(* IEC 61131-3 sources: AXOpen/src/integrations/app/src/Examples/AXOpen.AxoData, 8 files *)

(* ---- AxoDataDocuExample.st ---- *)
USING AXOpen.Core;
using AXOpen.Data;

NAMESPACE AxoDataExamplesDocu

    //<ProcessDataMangerDeclaration>
    {S7.extern=ReadWrite}
    CLASS AxoProcessDataManager EXTENDS AXOpen.Data.AxoDataExchange
        VAR PUBLIC
            {#ix-generic:TOnline}
            {#ix-generic:TPlain as POCO}
            {#ix-attr:[AxoDataEntityAttribute]}
            Data       : AxoProductionData;    // <-  Manager will operate on this member.
        END_VAR
    END_CLASS
    //</ProcessDataMangerDeclaration>

    //<ProcessDataDeclaration>
    {S7.extern=ReadWrite}
    CLASS AxoProductionData EXTENDS AXOpen.Data.AxoDataEntity
        VAR PUBLIC
            {#ix-set:AttributeName = "Some string data"}
            SomeData : STRING;
            {#ix-set:AttributeName = "Some number"}
            SomeNumber : INT;
            {#ix-set:AttributeName = "Some boolean"}
            SomeBool : BOOL;
        END_VAR
    END_CLASS
    //</ProcessDataDeclaration>

    //<ContextDeclaration>
    {S7.extern=ReadWrite}
    CLASS PUBLIC Context EXTENDS AXOpen.Core.AxoContext
        VAR PUBLIC
            DataManager : AxoProcessDataManager;
            _rootObject :   AxoObject;
        END_VAR

        METHOD OVERRIDE Main
            THIS.InitializeRootObject(_rootObject);
            DataManager.Run(_rootObject);
        END_METHOD
    END_CLASS
    //</ContextDeclaration>

    //<UseManager>
    {S7.extern=ReadWrite}
    CLASS UseManager
        VAR
            _create : BOOL;
            _read : BOOL;
            _update : BOOL;
            _delete : BOOL;
            _id : STRING;
        END_VAR

        METHOD Use
            VAR_IN_OUT
                DataManager : AxoProcessDataManager;
            END_VAR
            IF(_create) THEN
                IF(DataManager.Create(_id).IsDone()) THEN
                    _create := FALSE;
                END_IF;
            END_IF;

            IF(_read) THEN
                IF(DataManager.Read(_id).IsDone()) THEN
                    _read := FALSE;
                END_IF;
            END_IF;

            IF(_update) THEN
                IF(DataManager.Update(_id).IsDone()) THEN
                    _update := FALSE;
                END_IF;
            END_IF;

            IF(_delete) THEN
                IF(DataManager.Delete(_id).IsDone()) THEN
                    _delete := FALSE;
                END_IF;
            END_IF;
        END_METHOD
    END_CLASS
    //</UseManager>

END_NAMESPACE

(* ---- AxoDataFragmentExchangeDocu.st ---- *)
USING AXOpen.Core;
USING AXOpen.Data;
USING AXOpen.Probers;

NAMESPACE AxoDataFramentsExchangeDocuExample

    //<ContextDeclaration>
    {S7.extern=ReadWrite}
    CLASS AxoDataFragmentExchangeContext EXTENDS AXOpen.Core.AxoContext
        VAR PUBLIC
            ProcessData : ProcessDataManager;
            _rootObject :   AxoObject;
        END_VAR

        METHOD PROTECTED OVERRIDE Main
            _rootObject.InitializeWithContext(THIS);
            // This is required to run cyclically. Method provides handling of data exchange tasks.
            ProcessData.Run(_rootObject);
        END_METHOD
    END_CLASS
    //</ContextDeclaration>

    //<ProcessDataMangerDeclaration>
    {S7.extern=ReadWrite}
    CLASS ProcessDataManager EXTENDS AXOpen.Data.AxoDataFragmentExchange
        VAR PUBLIC
            {#ix-attr:[AXOpen.Data.AxoDataFragmentAttribute]}
            SharedHeader : SharedDataHeaderManger;
            {#ix-attr:[AXOpen.Data.AxoDataFragmentAttribute]}
            Station_1 : Station_1_ProcessDataManger;
        END_VAR
    END_CLASS
    //</ProcessDataMangerDeclaration>

     //<UseManager>
     {S7.extern=ReadWrite}
     CLASS UseManager
        VAR
            _create : BOOL;
            _read : BOOL;
            _update : BOOL;
            _delete : BOOL;
            _id : STRING;
        END_VAR

        METHOD Use
            VAR_IN_OUT
                DataFragmentManager : ProcessDataManager;
            END_VAR
            IF(_create) THEN
                IF(DataFragmentManager.Create(_id).IsDone()) THEN
                    _create := FALSE;
                END_IF;
            END_IF;

            IF(_read) THEN
                IF(DataFragmentManager.Read(_id).IsDone()) THEN
                    _read := FALSE;
                END_IF;
            END_IF;

            IF(_update) THEN
                IF(DataFragmentManager.Update(_id).IsDone()) THEN
                    _update := FALSE;
                END_IF;
            END_IF;

            IF(_delete) THEN
                IF(DataFragmentManager.Delete(_id).IsDone()) THEN
                    _delete := FALSE;
                END_IF;
            END_IF;
        END_METHOD
    END_CLASS
    //</UseManager>

    {S7.extern=ReadWrite}
    CLASS SharedDataHeaderData EXTENDS AXOpen.Data.AxoDataEntity
        VAR PUBLIC
            {#ix-set:AttributeName = "Some string data"}
            SomeData : STRING;
            {#ix-set:AttributeName = "Some number"}
            SomeNumber : INT;
            {#ix-set:AttributeName = "Some boolean"}
            SomeBool : BOOL;
        END_VAR
    END_CLASS

    {S7.extern=ReadWrite}
    CLASS SharedDataHeaderManger EXTENDS AXOpen.Data.AxoDataExchange
        VAR PUBLIC
            {#ix-generic:TOnline}
            {#ix-generic:TPlain as POCO}
            {#ix-attr:[AXOpen.Data.AxoDataEntityAttribute]}
            {#ix-attr:[Container(Layout.Stack)]}
            {#ix-set:AttributeName = "Shared Header"}
            Set : SharedDataHeaderData;
        END_VAR
    END_CLASS

    {S7.extern=ReadWrite}
    CLASS Station_1_ProcessDataManger
        EXTENDS AXOpen.Data.AxoDataExchange
        VAR PUBLIC
            {#ix-generic:TOnline}
            {#ix-generic:TPlain as POCO}
            {#ix-attr:[AXOpen.Data.AxoDataEntityAttribute]}
            {#ix-attr:[Container(Layout.Stack)]}
            {#ix-set:AttributeName = "Station 1"}
            Set : Station_1_Data;
        END_VAR
    END_CLASS

    {S7.extern=ReadWrite}
    CLASS Station_1_Data
        EXTENDS AXOpen.Data.AxoDataEntity
        VAR PUBLIC
            {#ix-set:AttributeName = "Some string data"}
            SomeData : STRING;
            {#ix-set:AttributeName = "Some number"}
            SomeNumber : INT;
            {#ix-set:AttributeName = "Some boolean"}
            SomeBool : BOOL;
        END_VAR
    END_CLASS
END_NAMESPACE

(* ---- AxoProcessDataManager.st ---- *)
using AXOpen.Data;

NAMESPACE AxoDataExamples

    CLASS AxoProcessDataManager EXTENDS AXOpen.Data.AxoDataExchange
        VAR PUBLIC
            _identifier : STRING;
            _create     : BOOL;
            _read       : BOOL;
            _update     : BOOL;
            _delete     : BOOL;
            {#ix-generic:TOnline}
            {#ix-generic:TPlain as POCO}
            {#ix-attr:[AxoDataEntityAttribute]}
            _data       : AxoProductionData;
            // _data       : AxoProductionDataInherited;
        END_VAR
    END_CLASS
END_NAMESPACE

(* ---- AxoProductionData.st ---- *)
using AXOpen.Data;

NAMESPACE AxoDataExamples

    CLASS AxoProductionData EXTENDS AXOpen.Data.AxoDataEntity
        VAR PUBLIC
            RecipeName : STRING;
        END_VAR
    END_CLASS

END_NAMESPACE

(* ---- AxoProductionDataInherited.st ---- *)
using AXOpen.Data;

NAMESPACE AxoDataExamples

    {S7.extern=ReadWrite}
    CLASS AxoProductionDataInherited EXTENDS AxoProductionData
        VAR PUBLIC
            RecipeName2 : STRING;
        END_VAR
    END_CLASS

END_NAMESPACE

(* ---- AxoTestData.st ---- *)
using AXOpen.Data;

NAMESPACE AxoDataExamples

    {#ix-attr:[Container(Layout.Tabs)]}
    {S7.extern=ReadWrite}
    CLASS AxoTestData EXTENDS AXOpen.Data.AxoDataEntity
        VAR PUBLIC
            RecipeName : STRING;
            String1 : STRING;
            Int1 : INT;
            Bool1 : BOOL;
            String2 : STRING;
            Int2 : INT;
            Bool2 : BOOL;
            String3 : STRING;
            Int3 : INT;
            Bool3 : BOOL;
            TestDataStructude : AxoTestDataStructure;
            {#ix-attr:[Container(Layout.UniformGrid)]}
            TestDataStructude2 : AxoTestDataStructure;
            {#ix-attr:[Container(Layout.Stack)]}
            TestDataStructude3 : AxoTestDataStructure;
            {#ix-attr:[Container(Layout.Wrap)]}
            TestDataStructude4 : AxoTestDataStructure;
        END_VAR
    END_CLASS

END_NAMESPACE

(* ---- AxoTestDataManager.st ---- *)
using AXOpen.Data;

NAMESPACE AxoDataExamples

    {S7.extern=ReadWrite}
    CLASS AxoTestDataManager EXTENDS AXOpen.Data.AxoDataExchange
        VAR PUBLIC
            _identifier : STRING;
            _create     : BOOL;
            _read       : BOOL;
            _update     : BOOL;
            _delete     : BOOL;
            {#ix-generic:TOnline}
            {#ix-generic:TPlain as POCO}
            {#ix-attr:[AxoDataEntityAttribute]}
            _data       : AxoTestData;
        END_VAR
    END_CLASS
END_NAMESPACE

(* ---- AxoTestDataStructure.st ---- *)
using AXOpen.Data;

NAMESPACE AxoDataExamples

    {S7.extern=ReadWrite}
    CLASS AxoTestDataStructure
        VAR PUBLIC
            RecipeName : STRING;
            String1 : STRING;
            Int1 : INT;
            Bool1 : BOOL;
            String2 : STRING;
            Int2 : INT;
            Bool2 : BOOL;
            String3 : STRING;
            Int3 : INT;
            Bool3 : BOOL;
        END_VAR
    END_CLASS
END_NAMESPACE
